{attribute addProperty BoxType "EP2339-0022-0016"}
{attribute addProperty Id "ChannelAT %I*ARRAY[0..15] OF Channel_E4AEF59E128160Channel_1_1AT %Q*Channel_7F374EB0810Channel_2_1AT %Q*Channel_7F374EB0810Channel_3_1AT %Q*Channel_7F374EB0810Channel_4_1AT %Q*Channel_7F374EB0810Channel_5_1AT %Q*Channel_7F374EB0810Channel_6_1AT %Q*Channel_7F374EB0810Channel_7_1AT %Q*Channel_7F374EB0810Channel_8_1AT %Q*Channel_7F374EB0810Channel_9_1AT %Q*Channel_7F374EB0810Channel_10_1AT %Q*Channel_7F374EB0810Channel_11_1AT %Q*Channel_7F374EB0810Channel_12_1AT %Q*Channel_7F374EB0810Channel_13_1AT %Q*Channel_7F374EB0810Channel_14_1AT %Q*Channel_7F374EB0810Channel_15_1AT %Q*Channel_7F374EB0810Channel_16_1AT %Q*Channel_7F374EB0810WcStateAT %I*WcState_98A4DF7520.250InfoDataAT %I*InfoData_192954DE1620"}
{attribute addProperty CRC "3300598566"}
{attribute addProperty SizeInBites "274"}
{attribute addProperty SizeInBytes "34.25"}
TYPE EP2339_D59416F6 :
STRUCT
	{attribute addProperty Name "Channel"}
	Channel : ARRAY[0..15] OF Channel_E4AEF59E;
	{attribute addProperty Name "Channel_1_1"}
	Channel_1_1 : Channel_7F374EB0;
	{attribute addProperty Name "Channel_2_1"}
	Channel_2_1 : Channel_7F374EB0;
	{attribute addProperty Name "Channel_3_1"}
	Channel_3_1 : Channel_7F374EB0;
	{attribute addProperty Name "Channel_4_1"}
	Channel_4_1 : Channel_7F374EB0;
	{attribute addProperty Name "Channel_5_1"}
	Channel_5_1 : Channel_7F374EB0;
	{attribute addProperty Name "Channel_6_1"}
	Channel_6_1 : Channel_7F374EB0;
	{attribute addProperty Name "Channel_7_1"}
	Channel_7_1 : Channel_7F374EB0;
	{attribute addProperty Name "Channel_8_1"}
	Channel_8_1 : Channel_7F374EB0;
	{attribute addProperty Name "Channel_9_1"}
	Channel_9_1 : Channel_7F374EB0;
	{attribute addProperty Name "Channel_10_1"}
	Channel_10_1 : Channel_7F374EB0;
	{attribute addProperty Name "Channel_11_1"}
	Channel_11_1 : Channel_7F374EB0;
	{attribute addProperty Name "Channel_12_1"}
	Channel_12_1 : Channel_7F374EB0;
	{attribute addProperty Name "Channel_13_1"}
	Channel_13_1 : Channel_7F374EB0;
	{attribute addProperty Name "Channel_14_1"}
	Channel_14_1 : Channel_7F374EB0;
	{attribute addProperty Name "Channel_15_1"}
	Channel_15_1 : Channel_7F374EB0;
	{attribute addProperty Name "Channel_16_1"}
	Channel_16_1 : Channel_7F374EB0;
	{attribute addProperty Name "WcState"}
	WcState : WcState_98A4DF75;
	{attribute addProperty Name "InfoData"}
	InfoData : InfoData_192954DE;
END_STRUCT
END_TYPE

(* stored: Version 1.2.0.0, ProductVersion 3.1.4024.9
   DUT EP2339_D59416F6: Id {ed55dafd-b680-42f6-b298-169a9006a384} *)
